Fanuc KAREL source: kt00605.KL

-- PROVISIONAL review KL for V770-1; original PC SHA256 0a05be04e36dd6a2756cbd250911bff799cb12df6f40e2a090b05f079c4fa679
-- Incomplete behavior may be omitted. Consult companion uncertainty JSON. Do not deploy.
PROGRAM KT00605
%NOLOCKGROUP
VAR
  I1 : INTEGER
  I2 : INTEGER
  OUT : REAL
BEGIN
  -- UNRESOLVED_PC offsets 5-16; opcodes 2E,23
  -- UNRESOLVED_PC offsets 21-32; opcodes 2E,23
  -- UNRESOLVED_PC offsets 37-48; opcodes 2E,23
  -- UNRESOLVED_PC offsets 53-64; opcodes 2E,23
  -- UNRESOLVED_PC offsets 69-83; opcodes 21,51,64,23
  -- UNRESOLVED_PC offsets 88-92; opcodes 7F
END KT00605
